FUNCTION F_DegreesToRadians : LREAL
VAR_INPUT
    degrees : LREAL;
END_VAR

F_DegreesToRadians := degrees * PI / 180.0;

END_FUNCTION

(* stored: Version 1.1.0.1, ProductVersion 3.1.4024.0
   POU F_DegreesToRadians: Id {3d0a6c4b-52de-4f0a-92d1-6d4be1b0c7a3}, SpecialFunc None *)
